// TIA Portal V21 export
FUNCTION_BLOCK "MV3000LineAnimation"   // FB801, LAD
{ S7_Optimized_Access := 'FALSE' }
// stored: AutoNumber false, SetENOAutomatically false
   VAR_INPUT
      AlwaysTrue : Bool;
      AlwaysFalse : Bool;
      SecPulse : Bool;
      "Spare 1" : Bool;
      "Spare 2" : Bool;
      "Spare 3" : Bool;
      "Spare 4" : Bool;
      "Spare 5" : Bool;
   END_VAR
   VAR
      "Node 1" : "LineAnimationFb";
      "Node 2" : "LineAnimationFb";
      "Node 3" : "LineAnimationFb";
      "Node 4" : "LineAnimationFb";
      "Node 5" : "LineAnimationFb";
      "Node 6" : "LineAnimationFb";
      "Node 7" { S7_SetPoint := 'True'} : "LineAnimationFb";
      "Node 8" { S7_SetPoint := 'True'} : "LineAnimationFb";
      "Node 9" { S7_SetPoint := 'True'} : "LineAnimationFb";
      "Node 10" { S7_SetPoint := 'True'} : "LineAnimationFb";
      "Node 11" { S7_SetPoint := 'True'} : "LineAnimationFb";
      "Node 12" { S7_SetPoint := 'True'} : "LineAnimationFb";
      "Node 13" { S7_SetPoint := 'True'} : "LineAnimationFb";
      "Node 14" { S7_SetPoint := 'True'} : "LineAnimationFb";
      "Node 15" { S7_SetPoint := 'True'} : "LineAnimationFb";
      "Node 16" { S7_SetPoint := 'True'} : "LineAnimationFb";
      "Node 17" { S7_SetPoint := 'True'} : "LineAnimationFb";
      "Node 18" { S7_SetPoint := 'True'} : "LineAnimationFb";
      "Node 19" { S7_SetPoint := 'True'} : "LineAnimationFb";
      "Node 20" { S7_SetPoint := 'True'} : "LineAnimationFb";
      "Node 21" { S7_SetPoint := 'True'} : "LineAnimationFb";
      "Node 22" { S7_SetPoint := 'True'} : "LineAnimationFb";
      "Node 23" { S7_SetPoint := 'True'} : "LineAnimationFb";
      "Node 24" { S7_SetPoint := 'True'} : "LineAnimationFb";
      "Node 25" { S7_SetPoint := 'True'} : "LineAnimationFb";
      "Node 26" { S7_SetPoint := 'True'} : "LineAnimationFb";
      "Node 27" { S7_SetPoint := 'True'} : "LineAnimationFb";
      "Node 28" { S7_SetPoint := 'True'} : "LineAnimationFb";
      "Node 29" { S7_SetPoint := 'True'} : "LineAnimationFb";
      "Node 30" { S7_SetPoint := 'True'} : "LineAnimationFb";
      Node31 { S7_SetPoint := 'True'} : "LineAnimationFb";
      Node32 { S7_SetPoint := 'True'} : "LineAnimationFb";
      Node33 { S7_SetPoint := 'True'} : "LineAnimationFb";
      Node34 { S7_SetPoint := 'True'} : "LineAnimationFb";
   END_VAR
BEGIN

REGION Network 1: Cv01,Cv02, Cv10
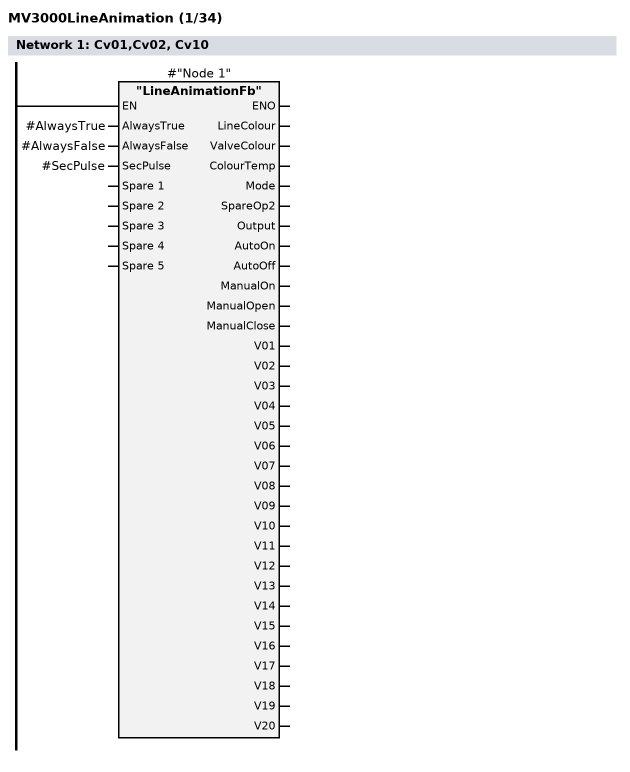
   RUNG wire#powerrail
      #"Node 1"(AlwaysTrue := #AlwaysTrue, AlwaysFalse := #AlwaysFalse, SecPulse := #SecPulse, "Spare 1" :=, "Spare 2" :=, "Spare 3" :=, "Spare 4" :=, "Spare 5" :=, LineColour =>, ValveColour =>, ColourTemp =>, Mode =>, SpareOp2 =>, Output =>, AutoOn =>, AutoOff =>, ManualOn =>, ManualOpen =>, ManualClose =>, V01 =>, V02 =>, V03 =>, V04 =>, V05 =>, V06 =>, V07 =>, V08 =>, V09 =>, V10 =>, V11 =>, V12 =>, V13 =>, V14 =>, V15 =>, V16 =>, V17 =>, V18 =>, V19 =>, V20 =>)
   END_RUNG
   // the same network as SCL:
   #"Node 1"(AlwaysTrue := #AlwaysTrue, AlwaysFalse := #AlwaysFalse, SecPulse := #SecPulse);   // "LineAnimationFb"
END_REGION

REGION Network 2: Cv03,Cv04,Cv05,Cv06
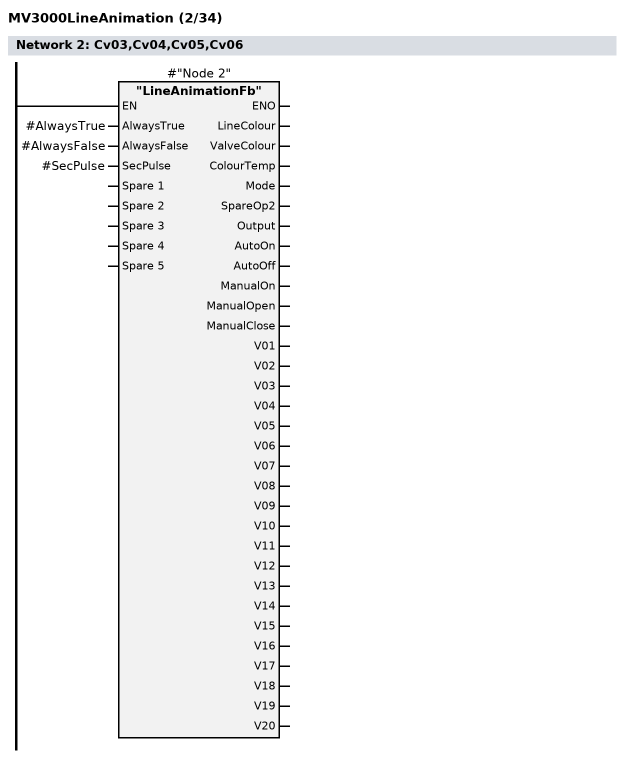
   RUNG wire#powerrail
      #"Node 2"(AlwaysTrue := #AlwaysTrue, AlwaysFalse := #AlwaysFalse, SecPulse := #SecPulse, "Spare 1" :=, "Spare 2" :=, "Spare 3" :=, "Spare 4" :=, "Spare 5" :=, LineColour =>, ValveColour =>, ColourTemp =>, Mode =>, SpareOp2 =>, Output =>, AutoOn =>, AutoOff =>, ManualOn =>, ManualOpen =>, ManualClose =>, V01 =>, V02 =>, V03 =>, V04 =>, V05 =>, V06 =>, V07 =>, V08 =>, V09 =>, V10 =>, V11 =>, V12 =>, V13 =>, V14 =>, V15 =>, V16 =>, V17 =>, V18 =>, V19 =>, V20 =>)
   END_RUNG
   // the same network as SCL:
   #"Node 2"(AlwaysTrue := #AlwaysTrue, AlwaysFalse := #AlwaysFalse, SecPulse := #SecPulse);   // "LineAnimationFb"
END_REGION

REGION Network 3: Cv07,Cv08, Cv09
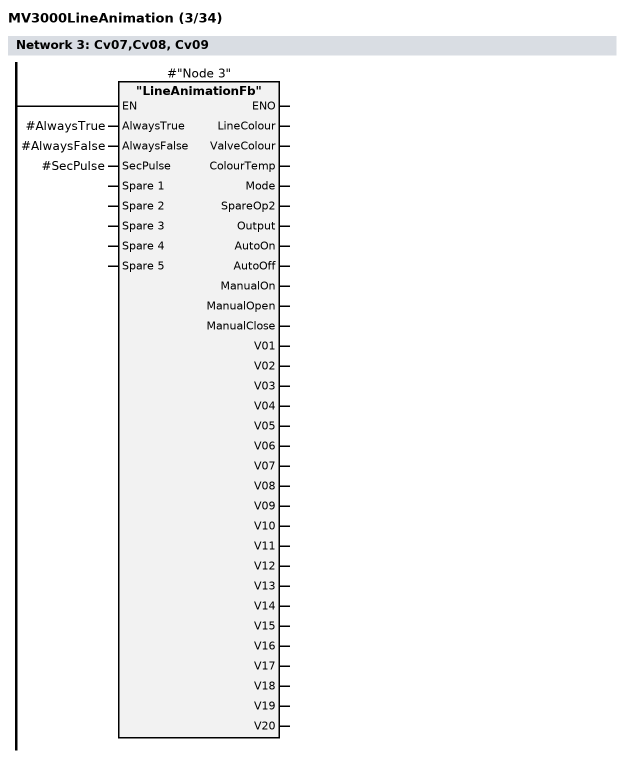
   RUNG wire#powerrail
      #"Node 3"(AlwaysTrue := #AlwaysTrue, AlwaysFalse := #AlwaysFalse, SecPulse := #SecPulse, "Spare 1" :=, "Spare 2" :=, "Spare 3" :=, "Spare 4" :=, "Spare 5" :=, LineColour =>, ValveColour =>, ColourTemp =>, Mode =>, SpareOp2 =>, Output =>, AutoOn =>, AutoOff =>, ManualOn =>, ManualOpen =>, ManualClose =>, V01 =>, V02 =>, V03 =>, V04 =>, V05 =>, V06 =>, V07 =>, V08 =>, V09 =>, V10 =>, V11 =>, V12 =>, V13 =>, V14 =>, V15 =>, V16 =>, V17 =>, V18 =>, V19 =>, V20 =>)
   END_RUNG
   // the same network as SCL:
   #"Node 3"(AlwaysTrue := #AlwaysTrue, AlwaysFalse := #AlwaysFalse, SecPulse := #SecPulse);   // "LineAnimationFb"
END_REGION

REGION Network 4: Cv16,Cv17,Cv22,Cv23,Cv24,Cv25
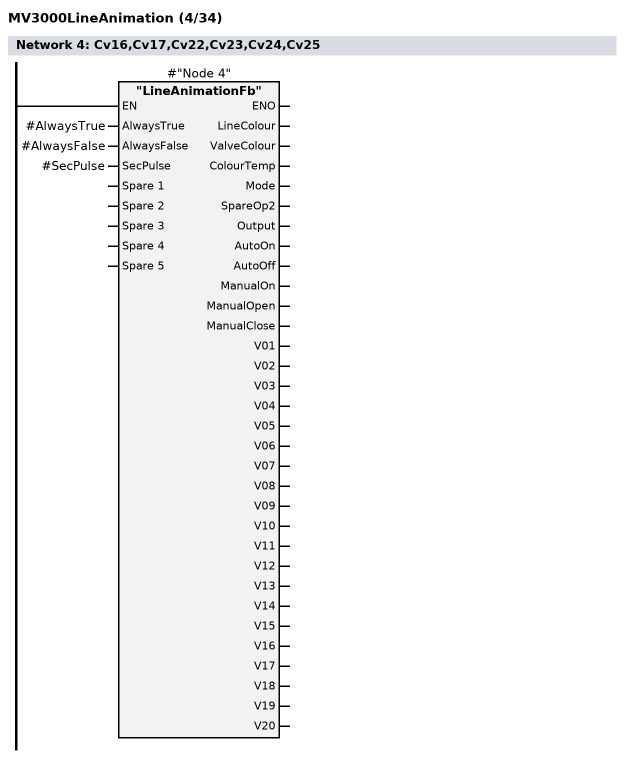
   RUNG wire#powerrail
      #"Node 4"(AlwaysTrue := #AlwaysTrue, AlwaysFalse := #AlwaysFalse, SecPulse := #SecPulse, "Spare 1" :=, "Spare 2" :=, "Spare 3" :=, "Spare 4" :=, "Spare 5" :=, LineColour =>, ValveColour =>, ColourTemp =>, Mode =>, SpareOp2 =>, Output =>, AutoOn =>, AutoOff =>, ManualOn =>, ManualOpen =>, ManualClose =>, V01 =>, V02 =>, V03 =>, V04 =>, V05 =>, V06 =>, V07 =>, V08 =>, V09 =>, V10 =>, V11 =>, V12 =>, V13 =>, V14 =>, V15 =>, V16 =>, V17 =>, V18 =>, V19 =>, V20 =>)
   END_RUNG
   // the same network as SCL:
   #"Node 4"(AlwaysTrue := #AlwaysTrue, AlwaysFalse := #AlwaysFalse, SecPulse := #SecPulse);   // "LineAnimationFb"
END_REGION

REGION Network 5: Cv22,Cv25
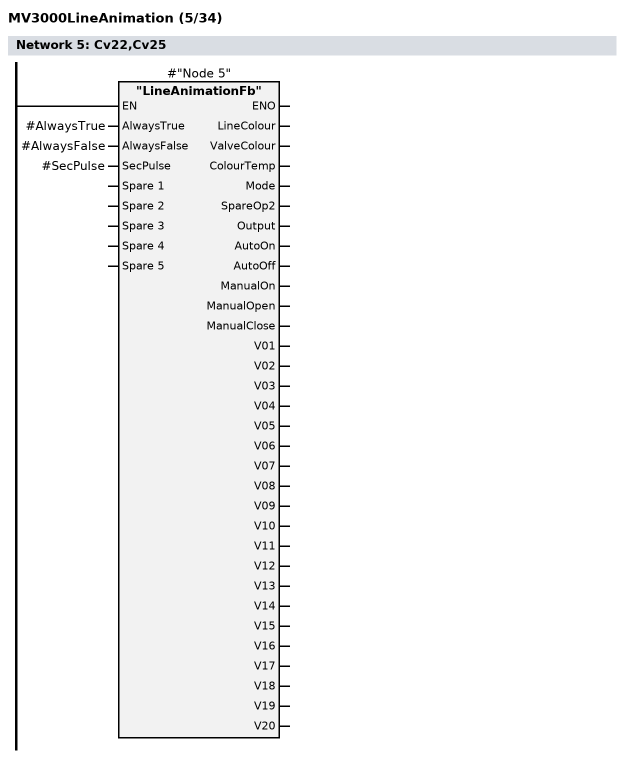
   RUNG wire#powerrail
      #"Node 5"(AlwaysTrue := #AlwaysTrue, AlwaysFalse := #AlwaysFalse, SecPulse := #SecPulse, "Spare 1" :=, "Spare 2" :=, "Spare 3" :=, "Spare 4" :=, "Spare 5" :=, LineColour =>, ValveColour =>, ColourTemp =>, Mode =>, SpareOp2 =>, Output =>, AutoOn =>, AutoOff =>, ManualOn =>, ManualOpen =>, ManualClose =>, V01 =>, V02 =>, V03 =>, V04 =>, V05 =>, V06 =>, V07 =>, V08 =>, V09 =>, V10 =>, V11 =>, V12 =>, V13 =>, V14 =>, V15 =>, V16 =>, V17 =>, V18 =>, V19 =>, V20 =>)
   END_RUNG
   // the same network as SCL:
   #"Node 5"(AlwaysTrue := #AlwaysTrue, AlwaysFalse := #AlwaysFalse, SecPulse := #SecPulse);   // "LineAnimationFb"
END_REGION

REGION Network 6: Cv18,Cv19,Cv20,Cv21
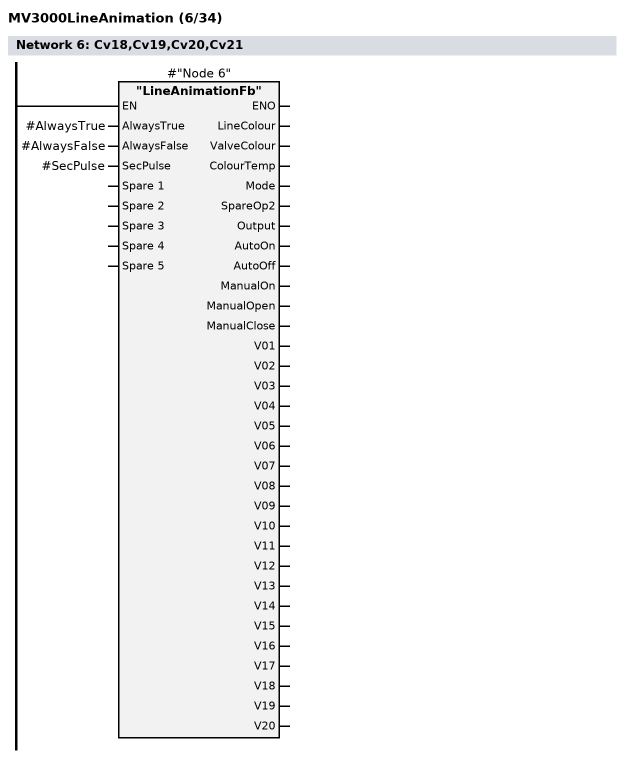
   RUNG wire#powerrail
      #"Node 6"(AlwaysTrue := #AlwaysTrue, AlwaysFalse := #AlwaysFalse, SecPulse := #SecPulse, "Spare 1" :=, "Spare 2" :=, "Spare 3" :=, "Spare 4" :=, "Spare 5" :=, LineColour =>, ValveColour =>, ColourTemp =>, Mode =>, SpareOp2 =>, Output =>, AutoOn =>, AutoOff =>, ManualOn =>, ManualOpen =>, ManualClose =>, V01 =>, V02 =>, V03 =>, V04 =>, V05 =>, V06 =>, V07 =>, V08 =>, V09 =>, V10 =>, V11 =>, V12 =>, V13 =>, V14 =>, V15 =>, V16 =>, V17 =>, V18 =>, V19 =>, V20 =>)
   END_RUNG
   // the same network as SCL:
   #"Node 6"(AlwaysTrue := #AlwaysTrue, AlwaysFalse := #AlwaysFalse, SecPulse := #SecPulse);   // "LineAnimationFb"
END_REGION

REGION Network 7: Cv19,Cv20
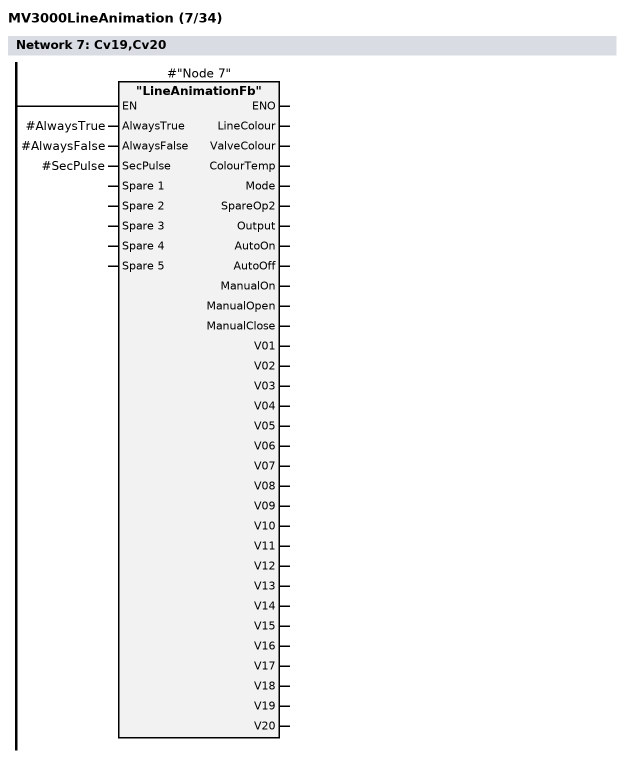
   RUNG wire#powerrail
      #"Node 7"(AlwaysTrue := #AlwaysTrue, AlwaysFalse := #AlwaysFalse, SecPulse := #SecPulse, "Spare 1" :=, "Spare 2" :=, "Spare 3" :=, "Spare 4" :=, "Spare 5" :=, LineColour =>, ValveColour =>, ColourTemp =>, Mode =>, SpareOp2 =>, Output =>, AutoOn =>, AutoOff =>, ManualOn =>, ManualOpen =>, ManualClose =>, V01 =>, V02 =>, V03 =>, V04 =>, V05 =>, V06 =>, V07 =>, V08 =>, V09 =>, V10 =>, V11 =>, V12 =>, V13 =>, V14 =>, V15 =>, V16 =>, V17 =>, V18 =>, V19 =>, V20 =>)
   END_RUNG
   // the same network as SCL:
   #"Node 7"(AlwaysTrue := #AlwaysTrue, AlwaysFalse := #AlwaysFalse, SecPulse := #SecPulse);   // "LineAnimationFb"
END_REGION

REGION Network 8: Cv16,Cv63, Cv15
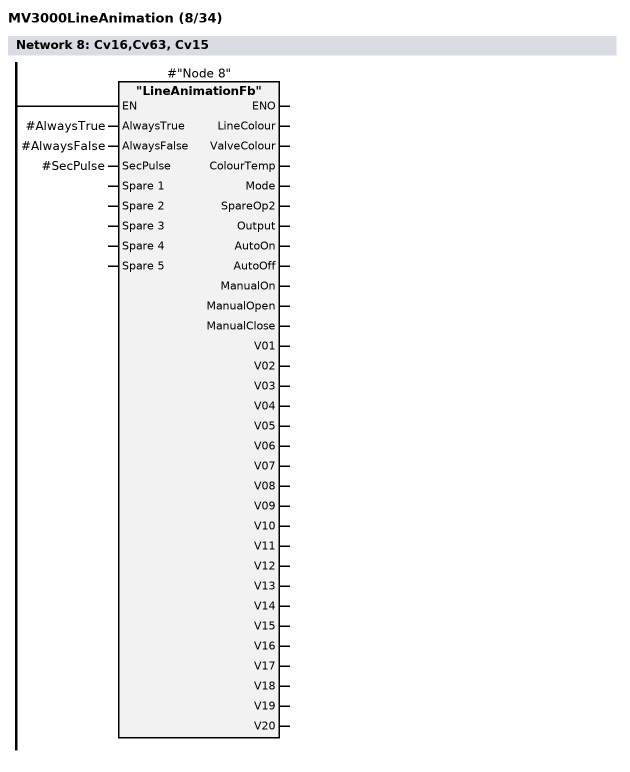
   RUNG wire#powerrail
      #"Node 8"(AlwaysTrue := #AlwaysTrue, AlwaysFalse := #AlwaysFalse, SecPulse := #SecPulse, "Spare 1" :=, "Spare 2" :=, "Spare 3" :=, "Spare 4" :=, "Spare 5" :=, LineColour =>, ValveColour =>, ColourTemp =>, Mode =>, SpareOp2 =>, Output =>, AutoOn =>, AutoOff =>, ManualOn =>, ManualOpen =>, ManualClose =>, V01 =>, V02 =>, V03 =>, V04 =>, V05 =>, V06 =>, V07 =>, V08 =>, V09 =>, V10 =>, V11 =>, V12 =>, V13 =>, V14 =>, V15 =>, V16 =>, V17 =>, V18 =>, V19 =>, V20 =>)
   END_RUNG
   // the same network as SCL:
   #"Node 8"(AlwaysTrue := #AlwaysTrue, AlwaysFalse := #AlwaysFalse, SecPulse := #SecPulse);   // "LineAnimationFb"
END_REGION

REGION Network 9: Cv10,Cv11,Cv12,Cv13,Cv14,Cv15
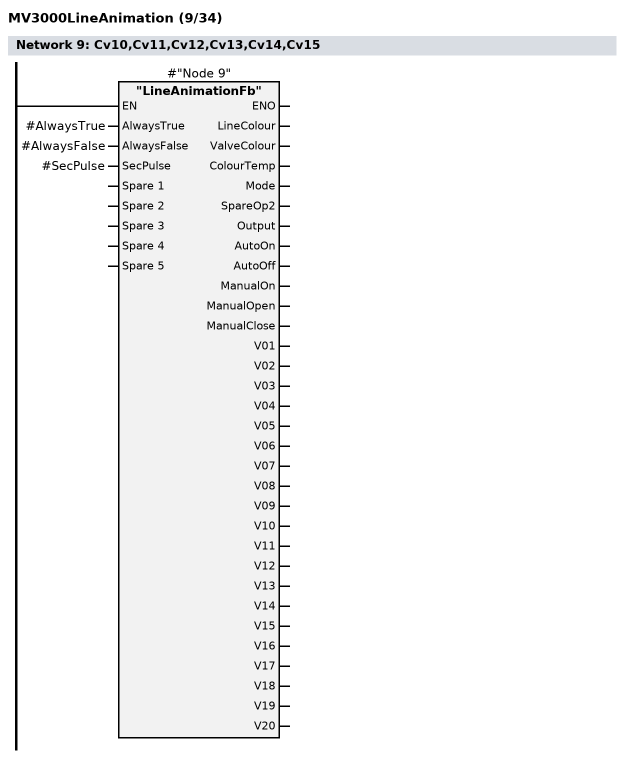
   RUNG wire#powerrail
      #"Node 9"(AlwaysTrue := #AlwaysTrue, AlwaysFalse := #AlwaysFalse, SecPulse := #SecPulse, "Spare 1" :=, "Spare 2" :=, "Spare 3" :=, "Spare 4" :=, "Spare 5" :=, LineColour =>, ValveColour =>, ColourTemp =>, Mode =>, SpareOp2 =>, Output =>, AutoOn =>, AutoOff =>, ManualOn =>, ManualOpen =>, ManualClose =>, V01 =>, V02 =>, V03 =>, V04 =>, V05 =>, V06 =>, V07 =>, V08 =>, V09 =>, V10 =>, V11 =>, V12 =>, V13 =>, V14 =>, V15 =>, V16 =>, V17 =>, V18 =>, V19 =>, V20 =>)
   END_RUNG
   // the same network as SCL:
   #"Node 9"(AlwaysTrue := #AlwaysTrue, AlwaysFalse := #AlwaysFalse, SecPulse := #SecPulse);   // "LineAnimationFb"
END_REGION

REGION Network 10: Cv11,Cv39
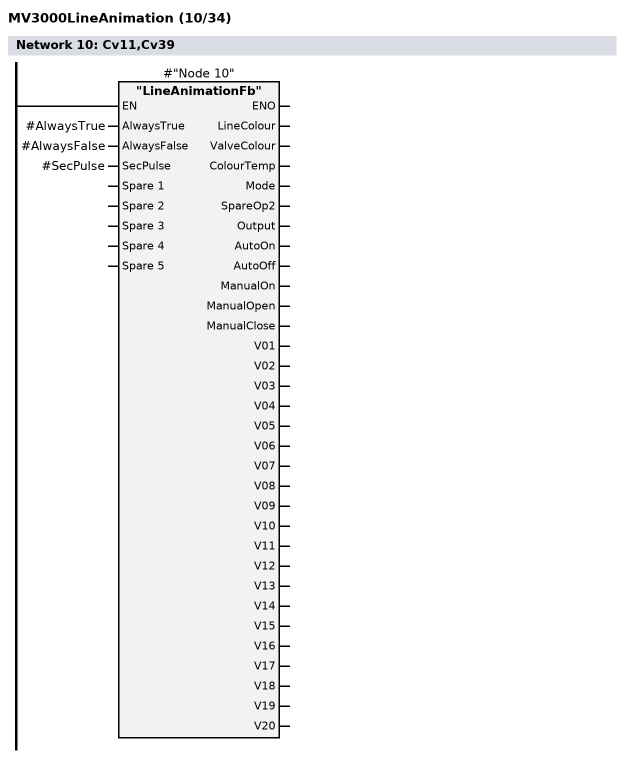
   RUNG wire#powerrail
      #"Node 10"(AlwaysTrue := #AlwaysTrue, AlwaysFalse := #AlwaysFalse, SecPulse := #SecPulse, "Spare 1" :=, "Spare 2" :=, "Spare 3" :=, "Spare 4" :=, "Spare 5" :=, LineColour =>, ValveColour =>, ColourTemp =>, Mode =>, SpareOp2 =>, Output =>, AutoOn =>, AutoOff =>, ManualOn =>, ManualOpen =>, ManualClose =>, V01 =>, V02 =>, V03 =>, V04 =>, V05 =>, V06 =>, V07 =>, V08 =>, V09 =>, V10 =>, V11 =>, V12 =>, V13 =>, V14 =>, V15 =>, V16 =>, V17 =>, V18 =>, V19 =>, V20 =>)
   END_RUNG
   // the same network as SCL:
   #"Node 10"(AlwaysTrue := #AlwaysTrue, AlwaysFalse := #AlwaysFalse, SecPulse := #SecPulse);   // "LineAnimationFb"
END_REGION

REGION Network 11: Cv12,Cv64, Cv26
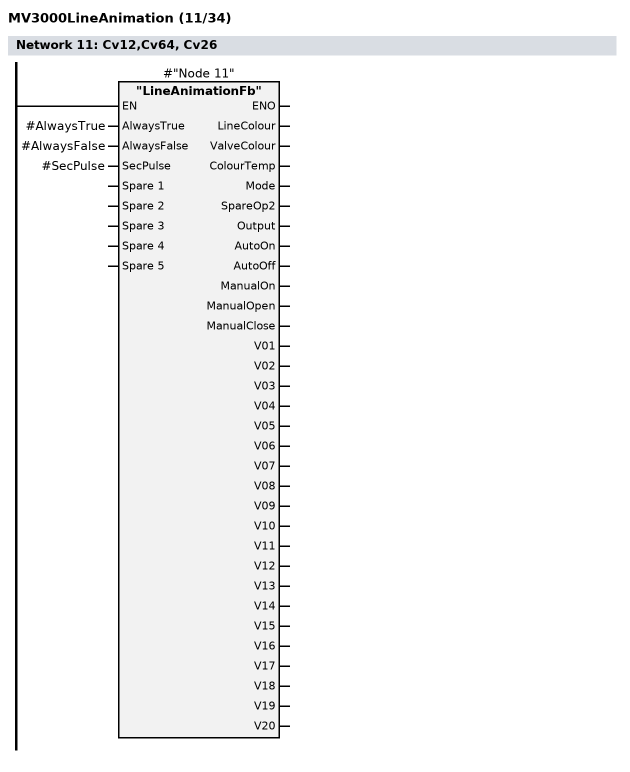
   RUNG wire#powerrail
      #"Node 11"(AlwaysTrue := #AlwaysTrue, AlwaysFalse := #AlwaysFalse, SecPulse := #SecPulse, "Spare 1" :=, "Spare 2" :=, "Spare 3" :=, "Spare 4" :=, "Spare 5" :=, LineColour =>, ValveColour =>, ColourTemp =>, Mode =>, SpareOp2 =>, Output =>, AutoOn =>, AutoOff =>, ManualOn =>, ManualOpen =>, ManualClose =>, V01 =>, V02 =>, V03 =>, V04 =>, V05 =>, V06 =>, V07 =>, V08 =>, V09 =>, V10 =>, V11 =>, V12 =>, V13 =>, V14 =>, V15 =>, V16 =>, V17 =>, V18 =>, V19 =>, V20 =>)
   END_RUNG
   // the same network as SCL:
   #"Node 11"(AlwaysTrue := #AlwaysTrue, AlwaysFalse := #AlwaysFalse, SecPulse := #SecPulse);   // "LineAnimationFb"
END_REGION

REGION Network 12: Cv31,Cv41
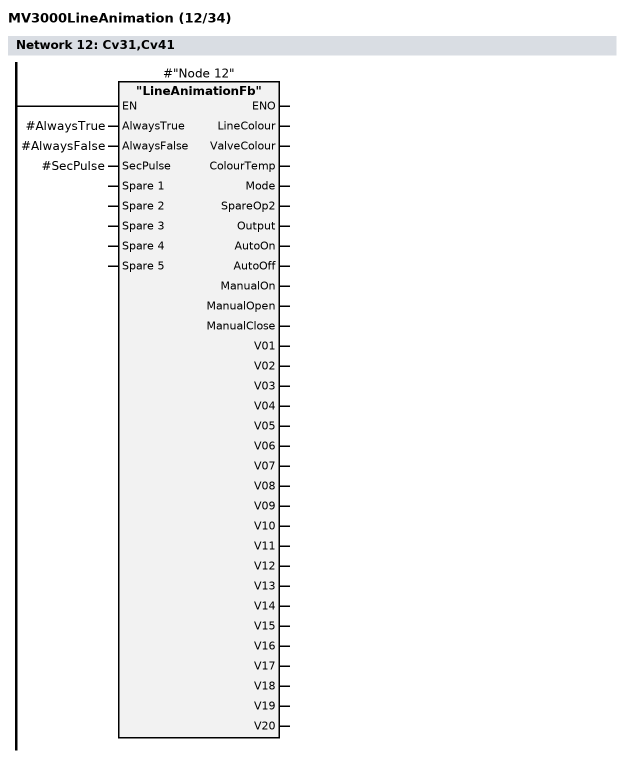
   RUNG wire#powerrail
      #"Node 12"(AlwaysTrue := #AlwaysTrue, AlwaysFalse := #AlwaysFalse, SecPulse := #SecPulse, "Spare 1" :=, "Spare 2" :=, "Spare 3" :=, "Spare 4" :=, "Spare 5" :=, LineColour =>, ValveColour =>, ColourTemp =>, Mode =>, SpareOp2 =>, Output =>, AutoOn =>, AutoOff =>, ManualOn =>, ManualOpen =>, ManualClose =>, V01 =>, V02 =>, V03 =>, V04 =>, V05 =>, V06 =>, V07 =>, V08 =>, V09 =>, V10 =>, V11 =>, V12 =>, V13 =>, V14 =>, V15 =>, V16 =>, V17 =>, V18 =>, V19 =>, V20 =>)
   END_RUNG
   // the same network as SCL:
   #"Node 12"(AlwaysTrue := #AlwaysTrue, AlwaysFalse := #AlwaysFalse, SecPulse := #SecPulse);   // "LineAnimationFb"
END_REGION

REGION Network 13: Fbov01, cV30 ,CV31 , CV 32 , CV33
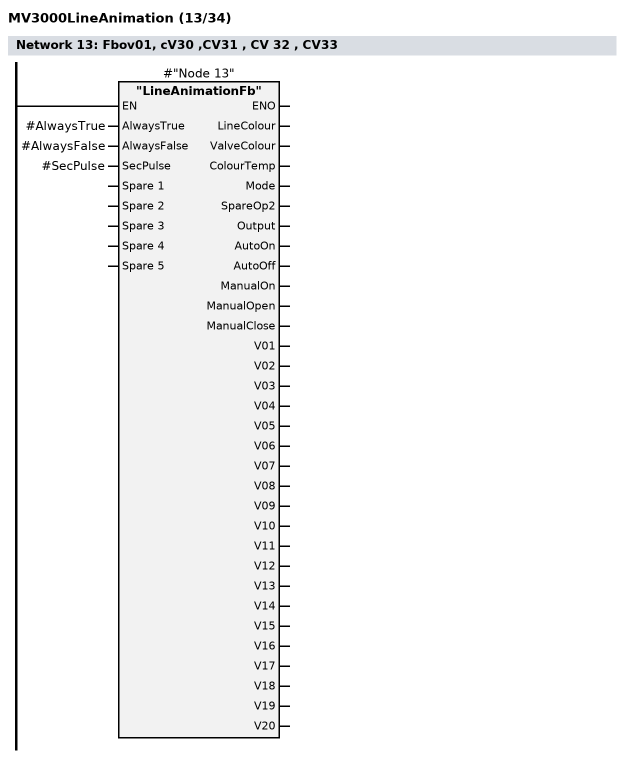
   RUNG wire#powerrail
      #"Node 13"(AlwaysTrue := #AlwaysTrue, AlwaysFalse := #AlwaysFalse, SecPulse := #SecPulse, "Spare 1" :=, "Spare 2" :=, "Spare 3" :=, "Spare 4" :=, "Spare 5" :=, LineColour =>, ValveColour =>, ColourTemp =>, Mode =>, SpareOp2 =>, Output =>, AutoOn =>, AutoOff =>, ManualOn =>, ManualOpen =>, ManualClose =>, V01 =>, V02 =>, V03 =>, V04 =>, V05 =>, V06 =>, V07 =>, V08 =>, V09 =>, V10 =>, V11 =>, V12 =>, V13 =>, V14 =>, V15 =>, V16 =>, V17 =>, V18 =>, V19 =>, V20 =>)
   END_RUNG
   // the same network as SCL:
   #"Node 13"(AlwaysTrue := #AlwaysTrue, AlwaysFalse := #AlwaysFalse, SecPulse := #SecPulse);   // "LineAnimationFb"
END_REGION

REGION Network 14: CV27 ,CV 28 ,CV 29
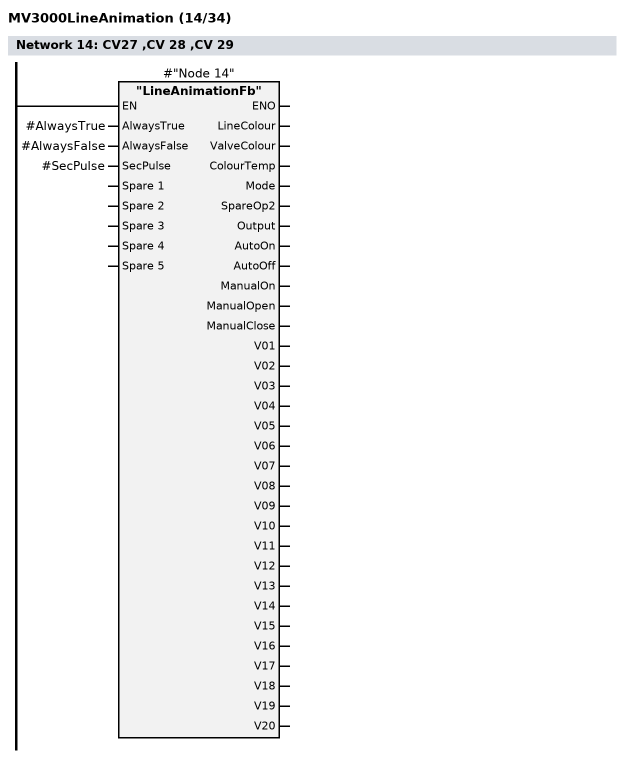
   RUNG wire#powerrail
      #"Node 14"(AlwaysTrue := #AlwaysTrue, AlwaysFalse := #AlwaysFalse, SecPulse := #SecPulse, "Spare 1" :=, "Spare 2" :=, "Spare 3" :=, "Spare 4" :=, "Spare 5" :=, LineColour =>, ValveColour =>, ColourTemp =>, Mode =>, SpareOp2 =>, Output =>, AutoOn =>, AutoOff =>, ManualOn =>, ManualOpen =>, ManualClose =>, V01 =>, V02 =>, V03 =>, V04 =>, V05 =>, V06 =>, V07 =>, V08 =>, V09 =>, V10 =>, V11 =>, V12 =>, V13 =>, V14 =>, V15 =>, V16 =>, V17 =>, V18 =>, V19 =>, V20 =>)
   END_RUNG
   // the same network as SCL:
   #"Node 14"(AlwaysTrue := #AlwaysTrue, AlwaysFalse := #AlwaysFalse, SecPulse := #SecPulse);   // "LineAnimationFb"
END_REGION

REGION Network 15: CV30 ,CV 33 ,CV 34,CV 35
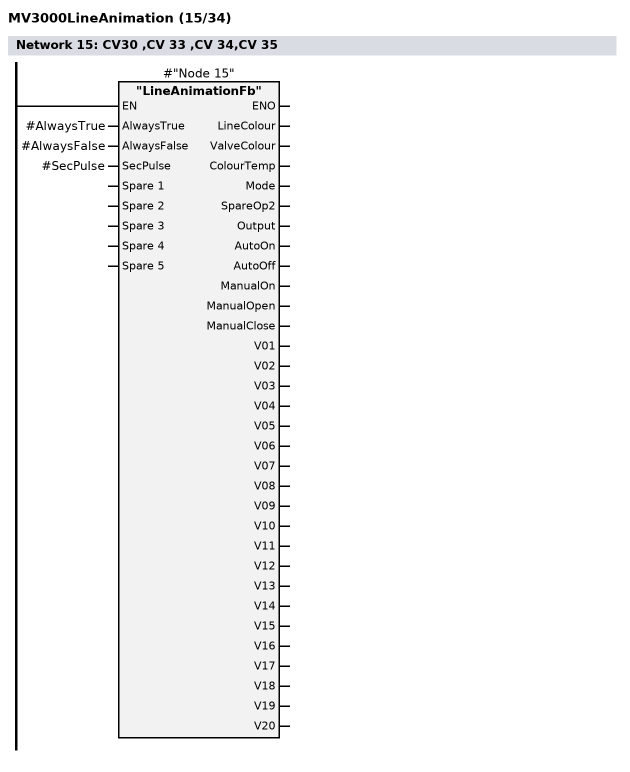
   RUNG wire#powerrail
      #"Node 15"(AlwaysTrue := #AlwaysTrue, AlwaysFalse := #AlwaysFalse, SecPulse := #SecPulse, "Spare 1" :=, "Spare 2" :=, "Spare 3" :=, "Spare 4" :=, "Spare 5" :=, LineColour =>, ValveColour =>, ColourTemp =>, Mode =>, SpareOp2 =>, Output =>, AutoOn =>, AutoOff =>, ManualOn =>, ManualOpen =>, ManualClose =>, V01 =>, V02 =>, V03 =>, V04 =>, V05 =>, V06 =>, V07 =>, V08 =>, V09 =>, V10 =>, V11 =>, V12 =>, V13 =>, V14 =>, V15 =>, V16 =>, V17 =>, V18 =>, V19 =>, V20 =>)
   END_RUNG
   // the same network as SCL:
   #"Node 15"(AlwaysTrue := #AlwaysTrue, AlwaysFalse := #AlwaysFalse, SecPulse := #SecPulse);   // "LineAnimationFb"
END_REGION

REGION Network 16: CV32 ,CV 36 ,CV 39,CV 40
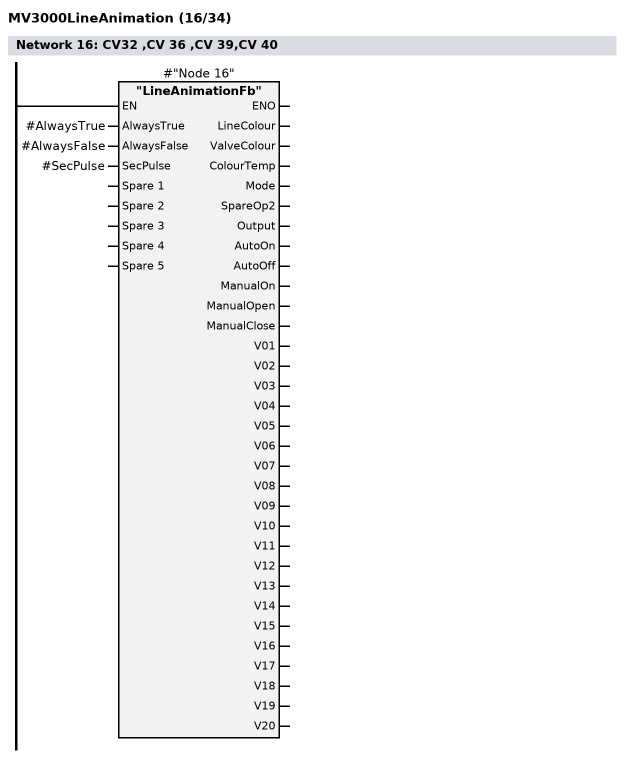
   RUNG wire#powerrail
      #"Node 16"(AlwaysTrue := #AlwaysTrue, AlwaysFalse := #AlwaysFalse, SecPulse := #SecPulse, "Spare 1" :=, "Spare 2" :=, "Spare 3" :=, "Spare 4" :=, "Spare 5" :=, LineColour =>, ValveColour =>, ColourTemp =>, Mode =>, SpareOp2 =>, Output =>, AutoOn =>, AutoOff =>, ManualOn =>, ManualOpen =>, ManualClose =>, V01 =>, V02 =>, V03 =>, V04 =>, V05 =>, V06 =>, V07 =>, V08 =>, V09 =>, V10 =>, V11 =>, V12 =>, V13 =>, V14 =>, V15 =>, V16 =>, V17 =>, V18 =>, V19 =>, V20 =>)
   END_RUNG
   // the same network as SCL:
   #"Node 16"(AlwaysTrue := #AlwaysTrue, AlwaysFalse := #AlwaysFalse, SecPulse := #SecPulse);   // "LineAnimationFb"
END_REGION

REGION Network 17: CV40 ,CV41 ,CV 42 ,CV 43,CV 44
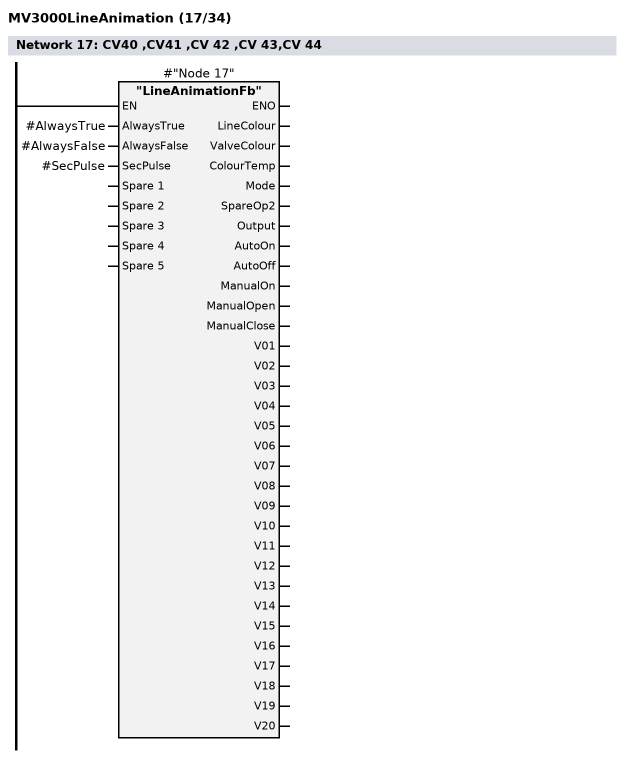
   RUNG wire#powerrail
      #"Node 17"(AlwaysTrue := #AlwaysTrue, AlwaysFalse := #AlwaysFalse, SecPulse := #SecPulse, "Spare 1" :=, "Spare 2" :=, "Spare 3" :=, "Spare 4" :=, "Spare 5" :=, LineColour =>, ValveColour =>, ColourTemp =>, Mode =>, SpareOp2 =>, Output =>, AutoOn =>, AutoOff =>, ManualOn =>, ManualOpen =>, ManualClose =>, V01 =>, V02 =>, V03 =>, V04 =>, V05 =>, V06 =>, V07 =>, V08 =>, V09 =>, V10 =>, V11 =>, V12 =>, V13 =>, V14 =>, V15 =>, V16 =>, V17 =>, V18 =>, V19 =>, V20 =>)
   END_RUNG
   // the same network as SCL:
   #"Node 17"(AlwaysTrue := #AlwaysTrue, AlwaysFalse := #AlwaysFalse, SecPulse := #SecPulse);   // "LineAnimationFb"
END_REGION

REGION Network 18: CV43 ,CV47 ,CV 48 ,CV 49,CV 50
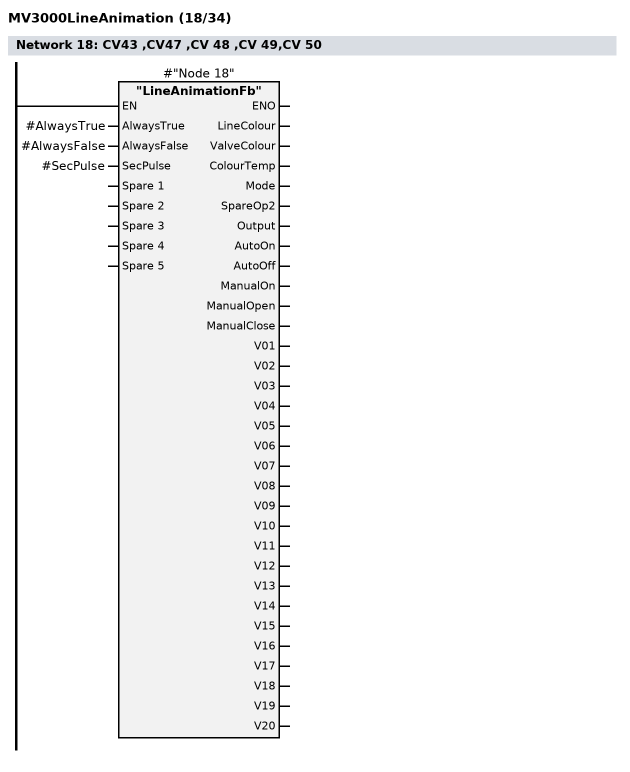
   RUNG wire#powerrail
      #"Node 18"(AlwaysTrue := #AlwaysTrue, AlwaysFalse := #AlwaysFalse, SecPulse := #SecPulse, "Spare 1" :=, "Spare 2" :=, "Spare 3" :=, "Spare 4" :=, "Spare 5" :=, LineColour =>, ValveColour =>, ColourTemp =>, Mode =>, SpareOp2 =>, Output =>, AutoOn =>, AutoOff =>, ManualOn =>, ManualOpen =>, ManualClose =>, V01 =>, V02 =>, V03 =>, V04 =>, V05 =>, V06 =>, V07 =>, V08 =>, V09 =>, V10 =>, V11 =>, V12 =>, V13 =>, V14 =>, V15 =>, V16 =>, V17 =>, V18 =>, V19 =>, V20 =>)
   END_RUNG
   // the same network as SCL:
   #"Node 18"(AlwaysTrue := #AlwaysTrue, AlwaysFalse := #AlwaysFalse, SecPulse := #SecPulse);   // "LineAnimationFb"
END_REGION

REGION Network 19: CV49 ,CV53 ,CV 54 ,CV 55,CV 56
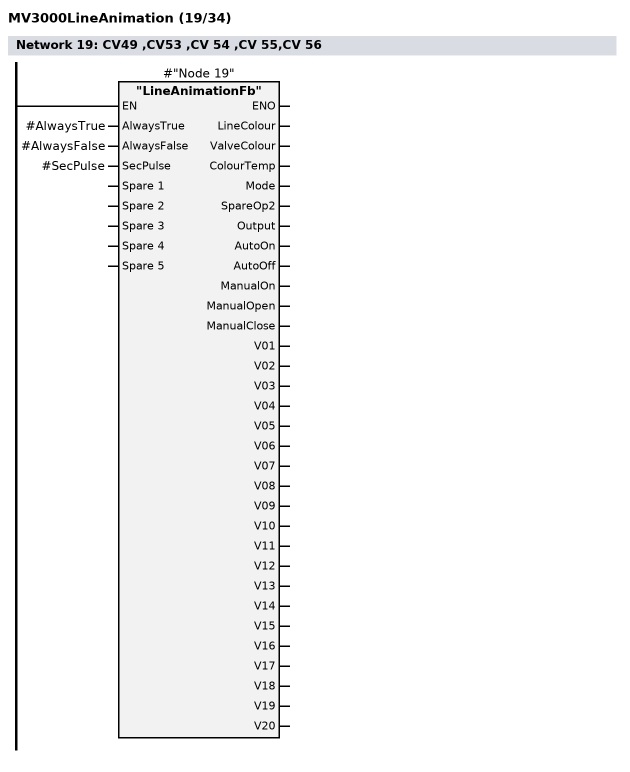
   RUNG wire#powerrail
      #"Node 19"(AlwaysTrue := #AlwaysTrue, AlwaysFalse := #AlwaysFalse, SecPulse := #SecPulse, "Spare 1" :=, "Spare 2" :=, "Spare 3" :=, "Spare 4" :=, "Spare 5" :=, LineColour =>, ValveColour =>, ColourTemp =>, Mode =>, SpareOp2 =>, Output =>, AutoOn =>, AutoOff =>, ManualOn =>, ManualOpen =>, ManualClose =>, V01 =>, V02 =>, V03 =>, V04 =>, V05 =>, V06 =>, V07 =>, V08 =>, V09 =>, V10 =>, V11 =>, V12 =>, V13 =>, V14 =>, V15 =>, V16 =>, V17 =>, V18 =>, V19 =>, V20 =>)
   END_RUNG
   // the same network as SCL:
   #"Node 19"(AlwaysTrue := #AlwaysTrue, AlwaysFalse := #AlwaysFalse, SecPulse := #SecPulse);   // "LineAnimationFb"
END_REGION

REGION Network 20: Cv55,Cv61, Cv62
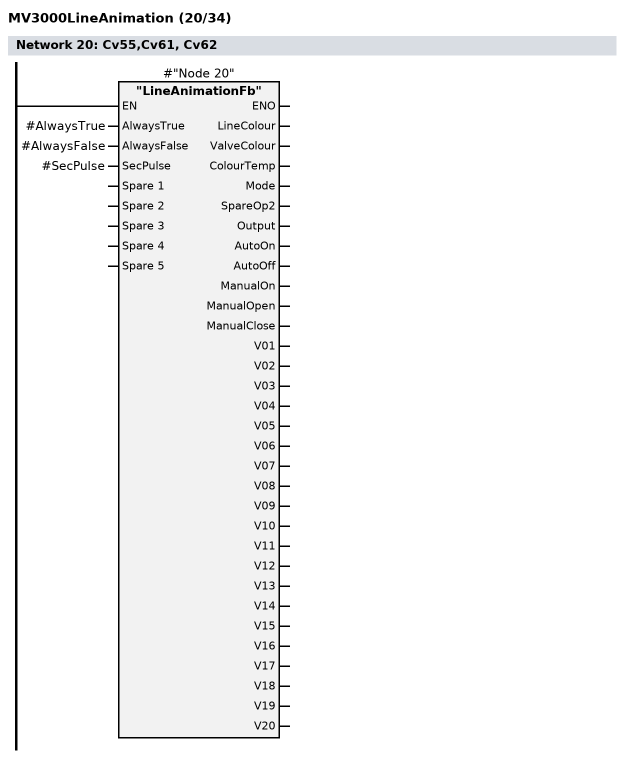
   RUNG wire#powerrail
      #"Node 20"(AlwaysTrue := #AlwaysTrue, AlwaysFalse := #AlwaysFalse, SecPulse := #SecPulse, "Spare 1" :=, "Spare 2" :=, "Spare 3" :=, "Spare 4" :=, "Spare 5" :=, LineColour =>, ValveColour =>, ColourTemp =>, Mode =>, SpareOp2 =>, Output =>, AutoOn =>, AutoOff =>, ManualOn =>, ManualOpen =>, ManualClose =>, V01 =>, V02 =>, V03 =>, V04 =>, V05 =>, V06 =>, V07 =>, V08 =>, V09 =>, V10 =>, V11 =>, V12 =>, V13 =>, V14 =>, V15 =>, V16 =>, V17 =>, V18 =>, V19 =>, V20 =>)
   END_RUNG
   // the same network as SCL:
   #"Node 20"(AlwaysTrue := #AlwaysTrue, AlwaysFalse := #AlwaysFalse, SecPulse := #SecPulse);   // "LineAnimationFb"
END_REGION

REGION Network 21: Cv59,Cv60, Cv61
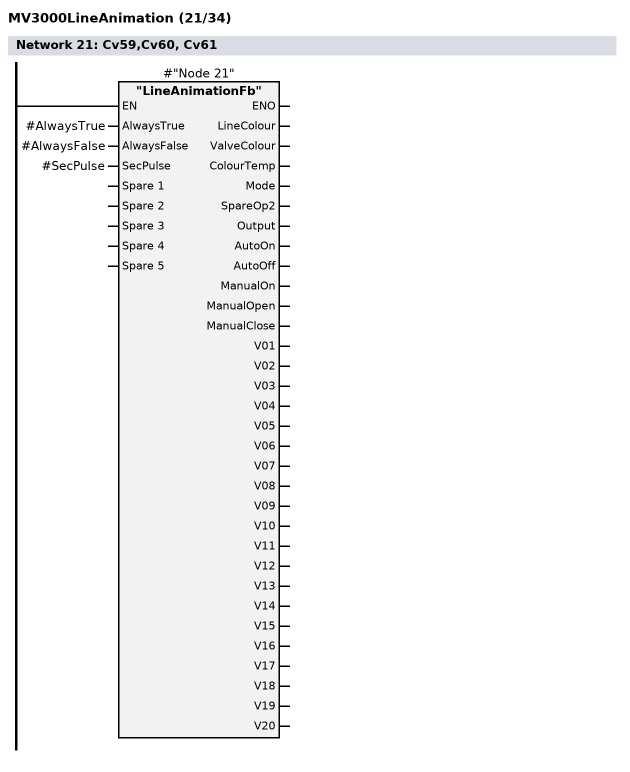
   RUNG wire#powerrail
      #"Node 21"(AlwaysTrue := #AlwaysTrue, AlwaysFalse := #AlwaysFalse, SecPulse := #SecPulse, "Spare 1" :=, "Spare 2" :=, "Spare 3" :=, "Spare 4" :=, "Spare 5" :=, LineColour =>, ValveColour =>, ColourTemp =>, Mode =>, SpareOp2 =>, Output =>, AutoOn =>, AutoOff =>, ManualOn =>, ManualOpen =>, ManualClose =>, V01 =>, V02 =>, V03 =>, V04 =>, V05 =>, V06 =>, V07 =>, V08 =>, V09 =>, V10 =>, V11 =>, V12 =>, V13 =>, V14 =>, V15 =>, V16 =>, V17 =>, V18 =>, V19 =>, V20 =>)
   END_RUNG
   // the same network as SCL:
   #"Node 21"(AlwaysTrue := #AlwaysTrue, AlwaysFalse := #AlwaysFalse, SecPulse := #SecPulse);   // "LineAnimationFb"
END_REGION

REGION Network 22: Cv56,Cv58, Cv57
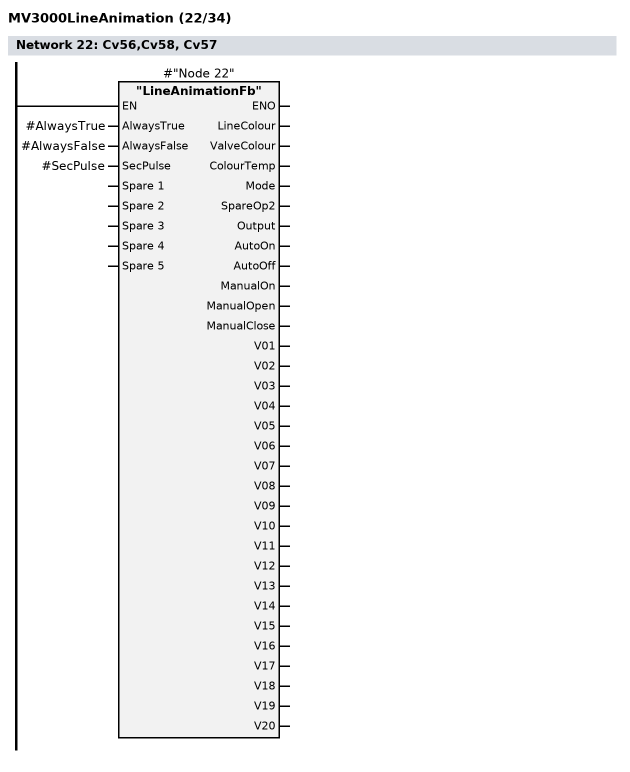
   RUNG wire#powerrail
      #"Node 22"(AlwaysTrue := #AlwaysTrue, AlwaysFalse := #AlwaysFalse, SecPulse := #SecPulse, "Spare 1" :=, "Spare 2" :=, "Spare 3" :=, "Spare 4" :=, "Spare 5" :=, LineColour =>, ValveColour =>, ColourTemp =>, Mode =>, SpareOp2 =>, Output =>, AutoOn =>, AutoOff =>, ManualOn =>, ManualOpen =>, ManualClose =>, V01 =>, V02 =>, V03 =>, V04 =>, V05 =>, V06 =>, V07 =>, V08 =>, V09 =>, V10 =>, V11 =>, V12 =>, V13 =>, V14 =>, V15 =>, V16 =>, V17 =>, V18 =>, V19 =>, V20 =>)
   END_RUNG
   // the same network as SCL:
   #"Node 22"(AlwaysTrue := #AlwaysTrue, AlwaysFalse := #AlwaysFalse, SecPulse := #SecPulse);   // "LineAnimationFb"
END_REGION

REGION Network 23: Cv50,Cv51, Cv52,Cv53
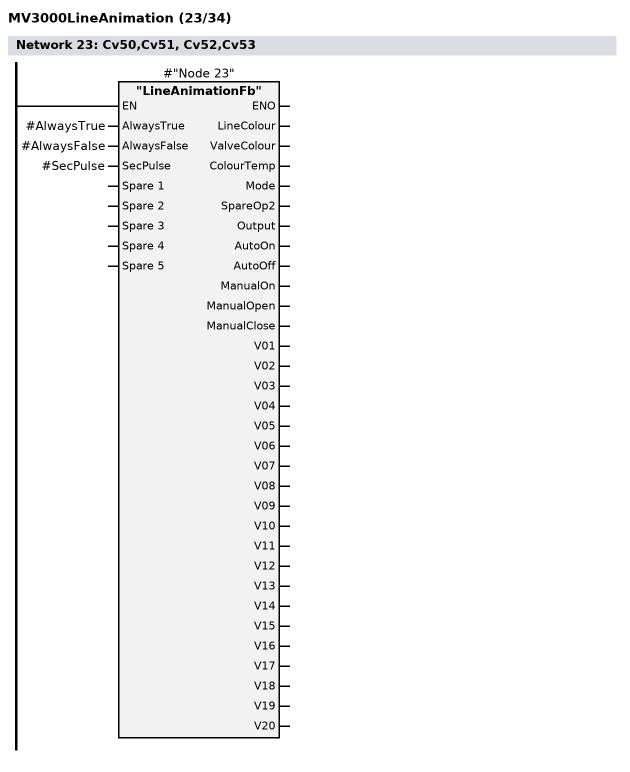
   RUNG wire#powerrail
      #"Node 23"(AlwaysTrue := #AlwaysTrue, AlwaysFalse := #AlwaysFalse, SecPulse := #SecPulse, "Spare 1" :=, "Spare 2" :=, "Spare 3" :=, "Spare 4" :=, "Spare 5" :=, LineColour =>, ValveColour =>, ColourTemp =>, Mode =>, SpareOp2 =>, Output =>, AutoOn =>, AutoOff =>, ManualOn =>, ManualOpen =>, ManualClose =>, V01 =>, V02 =>, V03 =>, V04 =>, V05 =>, V06 =>, V07 =>, V08 =>, V09 =>, V10 =>, V11 =>, V12 =>, V13 =>, V14 =>, V15 =>, V16 =>, V17 =>, V18 =>, V19 =>, V20 =>)
   END_RUNG
   // the same network as SCL:
   #"Node 23"(AlwaysTrue := #AlwaysTrue, AlwaysFalse := #AlwaysFalse, SecPulse := #SecPulse);   // "LineAnimationFb"
END_REGION

REGION Network 24: Cv44,Cv45, Cv46,Cv47
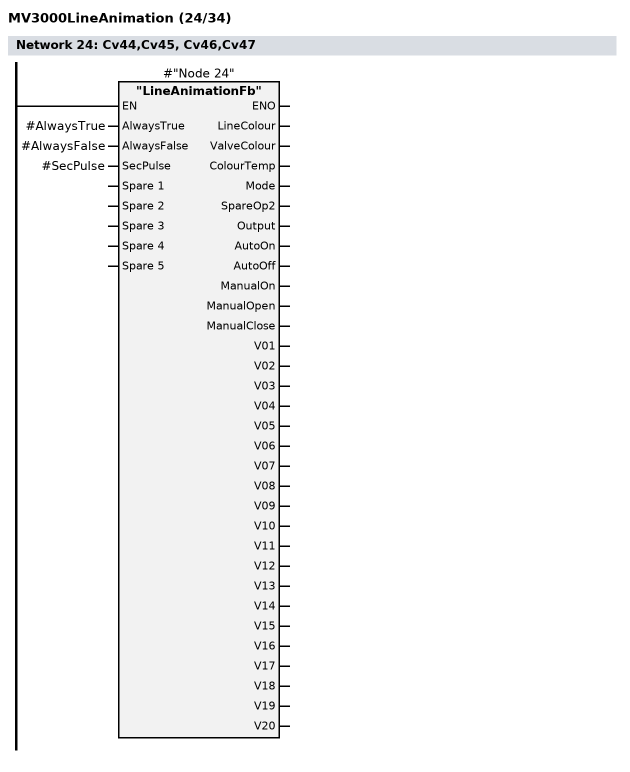
   RUNG wire#powerrail
      #"Node 24"(AlwaysTrue := #AlwaysTrue, AlwaysFalse := #AlwaysFalse, SecPulse := #SecPulse, "Spare 1" :=, "Spare 2" :=, "Spare 3" :=, "Spare 4" :=, "Spare 5" :=, LineColour =>, ValveColour =>, ColourTemp =>, Mode =>, SpareOp2 =>, Output =>, AutoOn =>, AutoOff =>, ManualOn =>, ManualOpen =>, ManualClose =>, V01 =>, V02 =>, V03 =>, V04 =>, V05 =>, V06 =>, V07 =>, V08 =>, V09 =>, V10 =>, V11 =>, V12 =>, V13 =>, V14 =>, V15 =>, V16 =>, V17 =>, V18 =>, V19 =>, V20 =>)
   END_RUNG
   // the same network as SCL:
   #"Node 24"(AlwaysTrue := #AlwaysTrue, AlwaysFalse := #AlwaysFalse, SecPulse := #SecPulse);   // "LineAnimationFb"
END_REGION

REGION Network 25: Cv36,Cv37, Cv38
